FUNCTION_BLOCK ChargeTimeCal
VAR_INPUT
	I_setpoint 	: REAL := 400;
	t_duration	: REAL := 4;
	NumOfCaps	: REAL := 15;
	C_percap	: REAL := 88;
	VMAXperCap	: REAL := 100;
	R_coil		: REAL := 1.1;
	L_coil		: REAL := 0.5;
	VMAXcharger	: REAL := 1500;
	Pcharger	: REAL := 15000;
	NumOfCharger: REAL := 4;
END_VAR
VAR_OUTPUT
	Tuntilfullcharge	: REAL;
END_VAR
VAR
	V_chargerCC2CP : REAL;
	C_total		   : REAL;
	V_capsmax	   : REAL;
	E_resistivepulse : REAL;
	E_inductivepulse : REAL;
	E_pulse			 : REAL;
	VchrSPrequested  : REAL;
	VchrSPactual     : REAL;
	I_peakchargecurrent : REAL;
	Icc					: REAL;
	Icp					: REAL;
	Vpresent			: REAL;
	Vfinal				: REAL;
	VpresentCC			: REAL;
	VfinalCC			: REAL;
	Tcc					: REAL;
	VpresentCP			: REAL;
	Tcp					: REAL;
END_VAR

V_chargerCC2CP := VMAXcharger / 2;

C_total := C_percap/NumOfCaps;
V_capsmax := VMAXpercap * NumOfCaps;
E_resistivepulse := LREAL_TO_REAL(EXPT(I_setpoint, 2))*R_coil*t_duration;
E_inductivepulse := L_coil * LREAL_TO_REAL(EXPT(I_setpoint, 2))/2;
E_pulse := E_resistivepulse + E_inductivepulse;
VchrSPrequested := SQRT(2*E_pulse/C_total);

IF VchrSPrequested > V_capsmax THEN
	VchrSPactual := V_capsmax;
	ELSE
		VchrSPactual := VchrSPrequested;	
END_IF

//I_peakchargecurrent := Pcharger * NumOfCharger / (2*VMAXcharger);
I_peakchargecurrent := Pcharger * NumOfCharger * 2 / VMAXcharger;
Icc := I_peakchargecurrent;
Icp := I_peakchargecurrent * (0.5 + ((VMAXcharger - Vpresent)/VMAXcharger));
Vfinal := 1400; //hard coded???
VpresentCC := 200; // hard coded???

IF Vfinal > V_chargerCC2CP THEN
	VfinalCC := V_chargerCC2CP;
	ELSIF Vfinal < V_chargerCC2CP THEN
		VfinalCC := Vfinal;
END_IF

Tcc := (V_chargerCC2CP - VpresentCC)*C_total/I_peakchargecurrent;

VpresentCP := V_chargerCC2CP;
Tcp := -((VMAXcharger*C_total)/I_peakchargecurrent)*LN((1.5*VMAXcharger-Vfinal)/(1.5*VMAXcharger-VpresentCP));

Tuntilfullcharge := Tcc + Tcp;

END_FUNCTION_BLOCK

(* stored: Version 1.1.0.1, ProductVersion 3.1.4024.11
   POU ChargeTimeCal: Id {2188ccf4-5a87-4717-accc-069ab0f00230}, SpecialFunc None *)
